(* IEC 61131-3 sources: example-modbus-rtu/PC WORX/export-st, 14 files *)

(* ---- sys_flag_types.IEC ---- *)
(*@PROPERTIES_EX@
TYPE: DATA_TYPE
LOCALE: 0
*)
TYPE
    Task_Name_Typ : ARRAY[0..9] OF BYTE;

    Extended_Task_Info : STRUCT
	    TaskName           : Task_Name_Typ;  (* Name of the Task as ARRAY OF BYTE, NULL terminated *)
	    TaskPrio           : INT;            (* Priority of the task *)
	    undocumented_0     : INT;
	    TaskPeriod         : INT;            (* Period of the task in milliseconds *)
	    TaskStack          : INT;            (* Stack size of the task *)
	    unused_1           : INT;
	    TaskWatchdog       : INT;            (* Watchdog time in milliseconds *)
	    undocumented_2     : INT;
	    undocumented_3     : INT;
	    undocumented_4     : INT;
	    CurDuration        : INT;            (* Current task duration in ticks including preemption *)
	    MinDuration        : INT;            (* Minimum task duration in ticks including preemption *)
	    MaxDuration        : INT;            (* Maximum task duration in ticks including preemption *)
	    undocumented_5     : INT;
	    CurDelay           : INT;            (* Current task delay in ticks including preemption *)
	    MinDelay           : INT;            (* Minimum task delay in ticks including preemption *)
	    MaxDelay           : INT;            (* Maximum task delay in ticks including preemption *)
    END_STRUCT;
END_TYPE

TYPE
	Task_Name_eCLR : ARRAY[0..35] OF BYTE;

	Task_Info_eCLR : STRUCT
		TaskStack       : INT;            (* Stack size of the task *)
		TaskPrio        : INT;            (* Priority of the task *)
		TaskPeriod_us   : DINT;           (* Period of the task in microseconds *)
		TaskWatchdog_us : DINT;           (* Watchdog time in microseconds *)
		TaskPeriod      : INT;            (* Period of the task in milliseconds *)
		TaskWatchdog    : INT;            (* Watchdog time in milliseconds *)
		MinDuration_us  : DINT;           (* Minimum task duration in microseconds including preemption *)
		MaxDuration_us  : DINT;           (* Maximum task duration in microseconds including preemption *)
		CurDuration_us  : DINT;           (* Current task duration in microseconds including preemption *)
		MinDelay_us     : DINT;           (* Minimum task delay in microseconds including preemption *)
		MaxDelay_us     : DINT;           (* Maximum task delay in microseconds including preemption *)
		CurDelay_us     : DINT;           (* Current task delay in microseconds including preemption *)
		MinDuration     : INT;            (* Minimum task duration in milliseconds including preemption *)
		MaxDuration     : INT;            (* Maximum task duration in milliseconds including preemption *)
		CurDuration     : INT;            (* Current task duration in milliseconds including preemption *)
		MinDelay        : INT;            (* Minimum task delay in milliseconds including preemption *)
		MaxDelay        : INT;            (* Maximum task delay in milliseconds including preemption *)
		CurDelay        : INT;            (* Current task delay in milliseconds including preemption *)
		unused_1        : DINT;
		unused_2        : DINT;
		unused_3        : DINT;
		unused_4        : DINT;
		unused_5        : DINT;
		unused_6        : DINT;
		unused_7        : DINT;
		unused_8        : DINT;
		unused_9        : DINT;
		TNameMaxSize    : INT;
		TNameSize       : INT;
		TaskName        : Task_Name_eCLR;
	END_STRUCT;
END_TYPE

TYPE
	PND_IO_6   : ARRAY[0..5]   OF BYTE;
	PND_IO_7   : ARRAY[0..6]   OF BYTE;
	PND_IO_32  : ARRAY[0..31]  OF BYTE;
	PND_IO_64  : ARRAY[0..63]  OF BYTE;
	PND_IO_128 : ARRAY[0..127] OF BYTE;
	PND_IO_256 : ARRAY[0..255] OF BYTE;
	PND_IO_512 : ARRAY[0..511] OF BYTE;
END_TYPE

TYPE
	Redundancy_OPC_Struct : ARRAY[0..2] OF INT;
END_TYPE

TYPE
    MBT_STATION_DIAG : STRUCT
	    Status           : DWORD; (* Bit 0 = Station is online*)
	                              (* Bit 1 = Exception exits  *)

	    IP               : DWORD;
	    OfflineCounter   : DWORD; (* Incremented by every shutdown of this station. *)

	    NetCycleAvg      : DWORD; (* ms. NetInCycleAvg + NetOutCycleAvg *)
	    NetCycleMin      : DWORD; (* ms. *)
	    NetCycleMax      : DWORD; (* ms. *)

	    NetInCycleAvg    : DWORD; (* ms. *)
	    NetInCycleMin    : DWORD; (* ms. *)
	    NetInCycleMax    : DWORD; (* ms. *)

	    NetOutCycleAvg   : DWORD; (* ms. *)
	    NetOutCycleMin   : DWORD; (* ms. *)
	    NetOutCycleMax   : DWORD; (* ms. *)

	    InternalError1   : DWORD; (* For internal use of Phoenix Contact! *)
	    InternalError2   : DWORD; (* For internal use of Phoenix Contact! *)

	    ExceptionCounter : DWORD; (* Incremented by every Modbus exception received on this station. *)
	    DiagReserved1    : BYTE;  (* Reserved for a later use! *)
	    DiagReserved2    : BYTE;  (* Reserved for a later use! *)
	    UnitID           : BYTE;  (* Modbus Unit Identifier *)
	    DiagReserved3    : BYTE;  (* Reserved for a later use! *)
    END_STRUCT;

    MBT_STATION_CONTROL : STRUCT
	    ctrlStatistics      : BYTE;  (* Bit 0 = Clear  statistics *)
	    ControlReserved1    : BYTE;  (* Reserved for a later use! *)
	    ControlReserved2    : WORD;  (* Reserved for a later use! *)
	    ControlReserved3    : DWORD; (* Reserved for a later use! *)
    END_STRUCT;
END_TYPE

TYPE
	MBS_SERVER_STATUS : STRUCT
		AcceptCnt              : DWORD;
		AcceptErrorCnt         : DWORD;
		ReceiveErrorCnt        : DWORD;
		ModbusRequestCnt       : DWORD;
		ModbusExceptionCnt     : DWORD;

		SocketErrorCode        : WORD;
		TcpConnectedClients    : WORD;
		LastExceptionRegister  : WORD;
		LastExceptionRegLength : WORD;

		LastExceptionNode      : BYTE;
		LastExceptionFunction  : BYTE;
		LastExceptionCode      : BYTE;
		reserved               : BYTE;
	END_STRUCT;
END_TYPE

TYPE
	MBS_SERVER_CONTROL : STRUCT
		Flags     : BYTE;
		reserved1 : BYTE;
		reserved2 : BYTE;
		reserved3 : BYTE;
	END_STRUCT;
END_TYPE

TYPE
	MBS_NODE_STATUS : STRUCT
		ModbusRequestCnt   : DWORD;
		ModbusExceptionCnt : DWORD;
		Flags              : DWORD;
		reserved           : DWORD;
	END_STRUCT;
END_TYPE

TYPE
    OPCUA_STATUS_INFO : STRUCT
	  restartCount            : UDINT; (* each reset and clear cache is counted *)
	  monitoredVariablesCount : UDINT; (* use IdataSource.GetSubscribedVariablesCount *)
	  sessionsCount           : UDINT; (* <-- get Data from ServerDiagnostic method GetTotalSubscribedVariablesCount *)
	  isServerEnabled         : UDINT; (* fetched by conf API *)
	  isLicensePresent        : UDINT; (* fetched by lic API *)
	END_STRUCT;
END_TYPE

TYPE
    IEC61850_TIMESTAMP : STRUCT
	    Seconds     : DWORD;
		Fractions   : DWORD;
        TimeQuality : DWORD;
    END_STRUCT;
END_TYPE

TYPE
	PROFISAFE_DIAG_HEADER : STRUCT
		NumberOfFConn         : UINT; (* number of F-Connections, max 256 *)
		PLCHostStatusByte     : BYTE; (* status byte of Standard PLC *)
		SPNSAgentStatusByte   : BYTE; (* status byte of SPNS agent *)
		CycleCount            : UINT;   (* cycle count off the spns agent (update the shm diag area) *)
	END_STRUCT;

	F_MESSAGE : ARRAY[0..15] OF BYTE; (* F-message: 16 bytes *)

	F_DEVICE_DIAG : STRUCT
		FAddress     : WORD;      (* F address of device  *)
		F_WD_Time    : WORD;      (* F WD time of device  *)
		F_DataLenIn  : BYTE;      (* length of IN F data  *)
		F_MessageIn  : F_MESSAGE; (* IN F data array      *)
		F_DataLenOut : BYTE;      (* length of OUT F data *)
		F_MessageOut : F_MESSAGE; (* OUT F data array     *)
	END_STRUCT;

	DEVICE_DIAG_LIST : ARRAY[0..255] OF F_DEVICE_DIAG; (* array of F_DEVICE_DIAG structurs: 256 elem *)

	PROFISAFE_DIAG : STRUCT
		ProfisafeDiagHeader : PROFISAFE_DIAG_HEADER; (* header *)
		FDeviceDiagnostics  : DEVICE_DIAG_LIST;      (* list of diagnostics *)
	END_STRUCT;
END_TYPE

TYPE
	PROFISAFE_RECORD : STRUCT
	   	CodeName              : DWORD;                   (* F_S/D_Address *)
   		ProfiSafeDiagBitField : DWORD;
   		SrtMin                : UINT;                    (* minimal safety round trip time of the connection *)
   		SrtMax                : UINT;                    (* maximal safety round trip time of the connection *)
   		SrtCur                : UINT;                    (* current safety round trip time of the connection *)
   		FWdTime               : UINT;                    (* parameterized f-wd-time *)
   		ValidReg              : UINT;                    (* the values in this profisafe record are balid or not *)
      	Reserved              : UINT;                    (* to fill up the structure to a size x*4 *)
 	END_STRUCT;

    PROFISAFE_RECORD_ARRAY : ARRAY[0..299] OF PROFISAFE_RECORD;

    PROFISAFE_DIAG_OUT : STRUCT
   		MaxNumberOfProfiSafeRecords : UINT; (* max. number of possible profisafe records *)
   		NumberOfProfiSafeRecords    : UINT; (* current number of possible profisafe records in array *)
   		ProfiSafeRecord             : PROFISAFE_RECORD_ARRAY;
   		ProfiSafeGlobalRecord       : DWORD;
 	END_STRUCT;
END_TYPE

(* ---- udtModbusControl.IEC ---- *)
(*@PROPERTIES_EX@
TYPE: DATA_TYPE
LOCALE: 0
*)
TYPE
	udtModbusControl	:
	STRUCT
		(* Commands to Modbus FB *)
		uiSlaveAddress		: UINT;

		xSendRequest_FC3	: BOOL;
		uiStartAddress_FC3	: UINT;
		iDataCount_FC3		: INT;

		xSendRequest_FC4	: BOOL;
		uiStartAddress_FC4	: UINT;
		iDataCount_FC4		: INT;

		xSendRequest_FC6	: BOOL;
		uiStartAddress_FC6	: UINT;

		(* Data from Modbus FB *)
		xDone_FC3			: BOOL;
		xError_FC3			: BOOL;
		arrReadData_FC3		: arrModbus2_W_1_125;

		xDone_FC4			: BOOL;
		xError_FC4			: BOOL;
		arrReadData_FC4		: arrModbus2_W_1_125;

		xDone_FC6			: BOOL;
		xError_FC6			: BOOL;
		wValue_FC6			: WORD;

		(* From udtMaster structure *)
		Master_uiRcvDataCount	: UINT;
		Master_uiSlaveAddress	: UINT;
		Master_uiStartAddress	: UINT;
		Master_iFunctionCode	: INT;
	END_STRUCT;
END_TYPE

(* ---- udtModbusDevice.IEC ---- *)
(*@PROPERTIES_EX@
TYPE: DATA_TYPE
LOCALE: 0
*)
TYPE
	udtModbusDiagValues:
	STRUCT
		xError							: BOOL;
		wDiagCode						: WORD;
		strDiagCode						: STRING;
	END_STRUCT;

	udtModbusConfiguration:
	STRUCT
		uiSlaveAddress					: UINT;
	END_STRUCT;

	udtDeviceConfiguration:
	STRUCT
		Modbus							: udtModbusConfiguration;
	END_STRUCT;

	udtDeviceDiagValues:
	STRUCT
		xError							: BOOL;
		wDiagCode						: WORD;
		strDiagCode						: STRING;

		Modbus							: udtModbusDiagValues;
	END_STRUCT;

	udtModbusDeviceValues:
	STRUCT
		iRtcMinutes						: INT;
	END_STRUCT;

	udtModbusDevice:
	STRUCT
		Configuration					: udtDeviceConfiguration;
		DataValues						: udtModbusDeviceValues;
		DiagValues						: udtDeviceDiagValues;
	END_STRUCT;
END_TYPE

(* ---- ErrorHandler.ST ---- *)
(*@PROPERTIES_EX@
TYPE: POU
LOCALE: 0
IEC_LANGUAGE: ST
PLC_TYPE: independent
PROC_TYPE: independent
GROUP: Modbus
*)
(*@KEY@:DESCRIPTION*)

(*@KEY@:END_DESCRIPTION*)
FUNCTION_BLOCK ErrorHandler

(*Group:Default*)

VAR_INPUT
	xError :	BOOL;
END_VAR

VAR
	wLastDiagCode :	WORD;
	wLastAddDiagCode :	WORD;
END_VAR

VAR_INPUT
	wDiagCode :	WORD;
	wAddDiagCode :	WORD;
END_VAR

(*@KEY@: WORKSHEET
NAME: ErrorHandler
IEC_LANGUAGE: ST
*)
IF xError THEN

	wLastDiagCode := wDiagCode;
	wLastAddDiagCode := wAddDiagCode;

END_IF;
(*@KEY@: END_WORKSHEET *)
END_FUNCTION_BLOCK

(* ---- MB_RTU_FC3_ABSTRACT.ST ---- *)
(*@PROPERTIES_EX@
TYPE: POU
LOCALE: 0
IEC_LANGUAGE: ST
PLC_TYPE: independent
PROC_TYPE: independent
GROUP: Modbus
*)
(*@KEY@:DESCRIPTION*)

(*@KEY@:END_DESCRIPTION*)
FUNCTION_BLOCK MB_RTU_FC3_ABSTRACT

(*Group:Input*)

VAR_INPUT
	xActivate :	BOOL;
	xSendRequest :	BOOL;
	xTimeout :	BOOL;
	uiSlaveAddress :	UINT;
	uiStartAddress :	UINT;
	iDataCount :	INT;
END_VAR

(*Group:Output*)

VAR_OUTPUT
	xDone :	BOOL;
	xError :	BOOL;
	xBusy :	BOOL;
	arrReadData :	arrModbus2_W_1_125;
END_VAR

(*Group:Inout*)

VAR_IN_OUT
	udtModbusControl :	udtModbusControl;
END_VAR

(*Group:Default*)

VAR
	iStep :	INT;
END_VAR

(*@KEY@: WORKSHEET
NAME: MB_RTU_FC3_ABSTRACT
IEC_LANGUAGE: ST
*)
IF xActivate THEN

	CASE iStep OF

		0:

			xDone	:= FALSE;
			xError	:= FALSE;

			IF xSendRequest THEN

				udtModbusControl.iDataCount_FC3 		:= iDataCount;
				udtModbusControl.uiSlaveAddress 		:= uiSlaveAddress;
				udtModbusControl.uiStartAddress_FC3		:= uiStartAddress;
				udtModbusControl.xSendRequest_FC3		:= TRUE;

				xBusy	:= TRUE;

				iStep := 1;

			END_IF;

		1:

	      udtModbusControl.xSendRequest_FC3     := FALSE;
		  udtModbusControl.iDataCount_FC3 		:= iDataCount;
		  udtModbusControl.uiSlaveAddress 		:= uiSlaveAddress;
		  udtModbusControl.uiStartAddress_FC3	:= uiStartAddress;

	      IF 	((udtModbusControl.xDone_FC3 OR
	        	udtModbusControl.xError_FC3) AND
	      		(udtModbusControl.Master_uiRcvDataCount = INT_TO_UINT(iDataCount * 2)) AND
	      		(udtModbusControl.Master_uiSlaveAddress  = uiSlaveAddress) AND
	      		(udtModbusControl.Master_uiStartAddress = uiStartAddress) AND
	      		(udtModbusControl.Master_iFunctionCode = 3))

				OR

				(*
				(xTimeout AND
				(udtModbusControl.Master_uiSlaveAddress  = uiSlaveAddress) AND
	      		(udtModbusControl.Master_uiStartAddress = uiStartAddress) AND
	      		(udtModbusControl.Master_iFunctionCode = 3))
				*)

				xTimeout

		  	THEN

					IF udtModbusControl.xDone_FC3 THEN
						arrReadData := udtModbusControl.arrReadData_FC3;
					END_IF;

					xDone	:= udtModbusControl.xDone_FC3;
					xError	:= udtModbusControl.xError_FC3 OR xTimeout;

					xBusy	:= FALSE;

					iStep := 0;

				END_IF;

	END_CASE;

ELSE

	xDone	:= FALSE;
	xError	:= FALSE;
	xBusy	:= FALSE;
	iStep	:= 0;

END_IF;

(*@KEY@: END_WORKSHEET *)
END_FUNCTION_BLOCK

(* ---- MB_RTU_FC4_ABSTRACT.ST ---- *)
(*@PROPERTIES_EX@
TYPE: POU
LOCALE: 0
IEC_LANGUAGE: ST
PLC_TYPE: independent
PROC_TYPE: independent
GROUP: Modbus
*)
(*@KEY@:DESCRIPTION*)

(*@KEY@:END_DESCRIPTION*)
FUNCTION_BLOCK MB_RTU_FC4_ABSTRACT

(*Group:Input*)

VAR_INPUT
	xActivate :	BOOL;
	xSendRequest :	BOOL;
	xTimeout :	BOOL;
	uiSlaveAddress :	UINT;
	uiStartAddress :	UINT;
	iDataCount :	INT;
END_VAR

(*Group:Output*)

VAR_OUTPUT
	xDone :	BOOL;
	xError :	BOOL;
	xBusy :	BOOL;
	arrReadData :	arrModbus2_W_1_125;
END_VAR

(*Group:Inout*)

VAR_IN_OUT
	udtModbusControl :	udtModbusControl;
END_VAR

(*Group:Default*)

VAR
	iStep :	INT;
END_VAR

(*@KEY@: WORKSHEET
NAME: MB_RTU_FC4_ABSTRACT
IEC_LANGUAGE: ST
*)
IF xActivate THEN

	CASE iStep OF

		0:

			xDone	:= FALSE;
			xError	:= FALSE;

			IF xSendRequest THEN

				udtModbusControl.iDataCount_FC4 		:= iDataCount;
				udtModbusControl.uiSlaveAddress 		:= uiSlaveAddress;
				udtModbusControl.uiStartAddress_FC4		:= uiStartAddress;
				udtModbusControl.xSendRequest_FC4		:= TRUE;

				xBusy	:= TRUE;

				iStep := 1;

			END_IF;

		1:

	      udtModbusControl.xSendRequest_FC4     := FALSE;
		  udtModbusControl.iDataCount_FC4 		:= iDataCount;
		  udtModbusControl.uiSlaveAddress 		:= uiSlaveAddress;
		  udtModbusControl.uiStartAddress_FC4	:= uiStartAddress;

	      IF 	((udtModbusControl.xDone_FC4 OR
	        	udtModbusControl.xError_FC4) AND
	      		(udtModbusControl.Master_uiRcvDataCount = INT_TO_UINT(iDataCount * 2)) AND
	      		(udtModbusControl.Master_uiSlaveAddress  = uiSlaveAddress) AND
	      		(udtModbusControl.Master_uiStartAddress = uiStartAddress) AND
	      		(udtModbusControl.Master_iFunctionCode = 4))

				OR

				(*
				(xTimeout AND
				(udtModbusControl.Master_uiSlaveAddress  = uiSlaveAddress) AND
	      		(udtModbusControl.Master_uiStartAddress = uiStartAddress) AND
	      		(udtModbusControl.Master_iFunctionCode = 3))
				*)

				xTimeout

		  	THEN

					IF udtModbusControl.xDone_FC4 THEN
						arrReadData := udtModbusControl.arrReadData_FC4;
					END_IF;

					xDone	:= udtModbusControl.xDone_FC4;
					xError	:= udtModbusControl.xError_FC4 OR xTimeout;

					xBusy	:= FALSE;

					iStep := 0;

				END_IF;

	END_CASE;

ELSE

	xDone	:= FALSE;
	xError	:= FALSE;
	xBusy	:= FALSE;
	iStep	:= 0;

END_IF;

(*@KEY@: END_WORKSHEET *)
END_FUNCTION_BLOCK

(* ---- MB_RTU_FC6_ABSTRACT.ST ---- *)
(*@PROPERTIES_EX@
TYPE: POU
LOCALE: 0
IEC_LANGUAGE: ST
PLC_TYPE: independent
PROC_TYPE: independent
GROUP: Modbus
*)
(*@KEY@:DESCRIPTION*)

(*@KEY@:END_DESCRIPTION*)
FUNCTION_BLOCK MB_RTU_FC6_ABSTRACT

(*Group:Default*)

VAR
	iStep :	INT;
END_VAR

(*Group:Input*)

VAR_INPUT
	xActivate :	BOOL;
	xSendRequest :	BOOL;
	xTimeout :	BOOL;
	uiSlaveAddress :	UINT;
	uiStartAddress :	UINT;
	wValue :	WORD;
END_VAR

(*Group:Output*)

VAR_OUTPUT
	xDone :	BOOL;
	xError :	BOOL;
	xBusy :	BOOL;
END_VAR

(*Group:Inout*)

VAR_IN_OUT
	udtModbusControl :	udtModbusControl;
END_VAR

(*@KEY@: WORKSHEET
NAME: MB_RTU_FC6_ABSTRACT
IEC_LANGUAGE: ST
*)
IF xActivate THEN

	CASE iStep OF

		0:

			xDone	:= FALSE;
			xError	:= FALSE;

			IF xSendRequest THEN

				udtModbusControl.uiSlaveAddress 		:= uiSlaveAddress;
				udtModbusControl.uiStartAddress_FC6		:= uiStartAddress;
				udtModbusControl.wValue_FC6				:= wValue;
				udtModbusControl.xSendRequest_FC6		:= TRUE;

				xBusy	:= TRUE;

				iStep := 1;

			END_IF;

		1:

			udtModbusControl.xSendRequest_FC6      := FALSE;
			udtModbusControl.uiSlaveAddress 		:= uiSlaveAddress;
			udtModbusControl.uiStartAddress_FC6		:= uiStartAddress;
			udtModbusControl.wValue_FC6				:= wValue;

			IF 	(
				(udtModbusControl.xDone_FC6 OR
	        	udtModbusControl.xError_FC6) AND
	      		(udtModbusControl.Master_uiSlaveAddress  = uiSlaveAddress) AND
	      		(udtModbusControl.Master_uiStartAddress = uiStartAddress) AND
	      		(udtModbusControl.Master_iFunctionCode = 6)
				)
				OR
				xTimeout

		  	THEN

					xDone	:= udtModbusControl.xDone_FC6;
					xError	:= udtModbusControl.xError_FC6 OR xTimeout;

					xBusy	:= FALSE;

					iStep := 0;

				END_IF;

	END_CASE;

ELSE

	xDone	:= FALSE;
	xError	:= FALSE;
	xBusy	:= FALSE;
	iStep	:= 0;

END_IF;

(*@KEY@: END_WORKSHEET *)
END_FUNCTION_BLOCK

(* ---- ModbusDeviceHandler.ST ---- *)
(*@PROPERTIES_EX@
TYPE: POU
LOCALE: 0
IEC_LANGUAGE: ST
PLC_TYPE: independent
PROC_TYPE: independent
GROUP: Modbus
*)
(*@KEY@:DESCRIPTION*)

(*@KEY@:END_DESCRIPTION*)
FUNCTION_BLOCK ModbusDeviceHandler

(*Group:POU`s*)

VAR
	TIME_DIFF :	TIME_DIFF;
	REQUEST_ERROR :	REQUEST_ERROR;
	MB_RTU_FC3_ABSTRACT :	MB_RTU_FC3_ABSTRACT;
END_VAR

(*Group:INTERNAL*)

VAR
	arrReadData_FC3 :	arrModbus2_W_1_125;
	xBusy_FC3 :	BOOL;
	xDone_FC3 :	BOOL;
	xError_FC3 :	BOOL;
	xTimeout_FC3 :	BOOL;
END_VAR

(*Group:INPUT*)

VAR_INPUT
	xActivate :	BOOL;
	xSendRequest_IN :	BOOL;
	uiSlaveAddress :	UINT;
END_VAR

(*Group:OUTPUT*)

VAR_OUTPUT
	xConnectionBroken :	BOOL;
	diTimeDiff :	DINT;
	xSendRequest_OUT :	BOOL;
END_VAR

(*Group:IN - OUT*)

VAR_INPUT
	ModbusDeviceData :	udtModbusDevice;
END_VAR

VAR_IN_OUT
	udtModbusControl :	udtModbusControl;
END_VAR

(*Group:Default*)

VAR_INPUT
	tTimeout :	TIME;
END_VAR

VAR
	RS_REQUEST_IN_PROGRESS :	RS;
END_VAR

(*@KEY@: WORKSHEET
NAME: ModbusDeviceHandler
IEC_LANGUAGE: ST
*)
(*	Request in progress *)
RS_REQUEST_IN_PROGRESS.SET					:= xActivate AND xSendRequest_IN;
RS_REQUEST_IN_PROGRESS.RESET1				:= NOT xActivate OR (xDone_FC3 OR xError_FC3);
RS_REQUEST_IN_PROGRESS();

(*	FC 3 *)
MB_RTU_FC3_ABSTRACT.xActivate				:= xActivate;
MB_RTU_FC3_ABSTRACT.xSendRequest			:= RS_REQUEST_IN_PROGRESS.Q1;
MB_RTU_FC3_ABSTRACT.xTimeout				:= xTimeout_FC3;
MB_RTU_FC3_ABSTRACT.uiSlaveAddress			:= uiSlaveAddress;
MB_RTU_FC3_ABSTRACT.uiStartAddress			:= UINT#1;
MB_RTU_FC3_ABSTRACT.iDataCount				:= INT#1;
MB_RTU_FC3_ABSTRACT.udtModbusControl		:= udtModbusControl;

MB_RTU_FC3_ABSTRACT();

xDone_FC3									:= MB_RTU_FC3_ABSTRACT.xDone;
xError_FC3									:= MB_RTU_FC3_ABSTRACT.xError;
xBusy_FC3									:= MB_RTU_FC3_ABSTRACT.xBusy;
arrReadData_FC3								:= MB_RTU_FC3_ABSTRACT.arrReadData;
udtModbusControl							:= MB_RTU_FC3_ABSTRACT.udtModbusControl;

(*	Pass the request to the next device handler *)
xSendRequest_OUT							:= RS_REQUEST_IN_PROGRESS.Q1 AND (xDone_FC3 OR xError_FC3);

(*	Detect errors *)
REQUEST_ERROR.xReq							:= xBusy_FC3;
REQUEST_ERROR.xDone							:= xDone_FC3;
REQUEST_ERROR.xError						:= xError_FC3;
REQUEST_ERROR.iMaxErrorCnt					:= 5;
REQUEST_ERROR.tTimeout						:= tTimeout;

REQUEST_ERROR();

xTimeout_FC3								:= REQUEST_ERROR.xTimeout;
ModbusDeviceData.DiagValues.Modbus.xError	:= REQUEST_ERROR.xConnectBroken;
xConnectionBroken							:= REQUEST_ERROR.xConnectBroken;

(*	Measure request time *)
TIME_DIFF.xIN1								:= xSendRequest_IN;
TIME_DIFF.xIN2								:= xSendRequest_OUT;
TIME_DIFF();
diTimeDiff									:= TIME_DIFF.diSystemTickDiff;

(*	Handle data values *)
ModbusDeviceData.DataValues.iRtcMinutes		:= WORD_TO_INT(arrReadData_FC3[1]);

(*	Handle diag values *)
IF ModbusDeviceData.DiagValues.Modbus.xError THEN

	ModbusDeviceData.DiagValues.xError		:=	TRUE;
	ModbusDeviceData.DiagValues.strDiagCode	:=	'RS-485 connection error';

ELSE
	ModbusDeviceData.DiagValues.xError		:=	FALSE;
	ModbusDeviceData.DiagValues.strDiagCode	:=	'OK';
END_IF;

(*@KEY@: END_WORKSHEET *)
END_FUNCTION_BLOCK

(* ---- REQ_CNT.ST ---- *)
(*@PROPERTIES_EX@
TYPE: POU
LOCALE: 0
IEC_LANGUAGE: ST
PLC_TYPE: independent
PROC_TYPE: independent
GROUP: Modbus
*)
(*@KEY@:DESCRIPTION*)
(*
FB generate a boolean output if:
	uiReqNo
	uiRespNo
do not counting up longer than specified delay time

*)
************
Versioning
************

15.01.2016	KONOPKOV Inital Version

(*@KEY@:END_DESCRIPTION*)
FUNCTION_BLOCK REQ_CNT

(*Group:outputs*)

VAR_OUTPUT
	xOut :	BOOL;
END_VAR

(*Group:internal*)

VAR
	uiReqNo_Registered :	UINT {RDT};
	uiRespNo_Registered :	UINT {RDT};
	TON_1 :	TON;
	TON_2 :	TON;
END_VAR

(*Group:inputs*)

VAR_INPUT
	xDisable :	BOOL;
	tTimeDelayRequests :	TIME;
	tTimeDelayResponces :	TIME;
	uiReqNo :	UINT;
	uiRespNo :	UINT;
END_VAR

VAR
	R_TRIG_1 :	R_TRIG;
END_VAR

(*@KEY@: WORKSHEET
NAME: REQ_CNT
IEC_LANGUAGE: ST
*)
(*
FB generate a boolean output if:
	uiReqNo
	uiRespNo
do not counting up longer than specified delay time

*)

TON_1.IN := (uiReqNo = uiReqNo_Registered AND NOT xDisable AND NOT xOut);
TON_1.PT := tTimeDelayRequests;
TON_1(); (*uiReqNo*)

TON_2.IN := (uiRespNo = uiRespNo_Registered AND NOT xDisable AND NOT xOut);
TON_2.PT := tTimeDelayResponces;
TON_2(); (*uiRespNo*)

R_TRIG_1.CLK 	:= TON_1.Q OR TON_2.Q;
R_TRIG_1();
xOut			:= R_TRIG_1.Q;

IF uiReqNo <> uiReqNo_Registered THEN
	uiReqNo_Registered := uiReqNo;
END_IF;

IF uiRespNo <> uiRespNo_Registered THEN
	uiRespNo_Registered := uiRespNo;
END_IF;

(*@KEY@: END_WORKSHEET *)
END_FUNCTION_BLOCK

(* ---- REQUEST_ERROR.ST ---- *)
(*@PROPERTIES_EX@
TYPE: POU
LOCALE: 0
IEC_LANGUAGE: ST
PLC_TYPE: independent
PROC_TYPE: independent
GROUP: Modbus
*)
(*@KEY@:DESCRIPTION*)
**************************************************************************

Copyright © 2016 Phoenix Contact Russia
All rights reserved

**************************************************************************
Name	:	 REQUEST_ERROR

State	:	[ ] evaluation  [x] released

Develop Environment	:
	PC WORX 	:	6.30.1668 (AX SW Suite 2016 Hotfix1)
	Controller	:	AXC 1050 FW v2.10
	Devices		: 	No

**************************************************************************

Change Notes:

Date		Version		Author		Description
--------------------------------------------------------------------------
08.08.16	1.00		konopkov	initial version

**************************************************************************
Description:
Индикация ошибки отсутствия обмена данными при достижении заданного количества
импульсов на вход Ошибка.

(*@KEY@:END_DESCRIPTION*)
FUNCTION_BLOCK REQUEST_ERROR

(*Group:Input*)

VAR_INPUT
	xReq :	BOOL;(*???? ??????*)
	xDone :	BOOL;(*???? ????? ??*)
	xError :	BOOL;(*???? ????? ??????*)
	iMaxErrorCnt :	INT := 5;(*???????????? ?????????? ????????? ?????? ? ??????????? ??????????????????*)
	tTimeout :	TIME;
END_VAR

(*Group:Output*)

VAR_OUTPUT
	xConnectBroken :	BOOL;(*??????? ??????????????? ?????? ?????*)
	xTimeout :	BOOL;
END_VAR

(*Group:Internal*)

VAR_OUTPUT
	iErrorCnt :	INT;(*??????? ??????*)
END_VAR

(*Group:Instances*)

VAR
	R_TRIG_DONE :	R_TRIG;
	R_TRIG_ERROR :	R_TRIG;
	R_TRIG_REQUEST :	R_TRIG;
	RS_REQUEST :	RS;
	TON_REQUEST :	TON;
END_VAR

(*@KEY@: WORKSHEET
NAME: REQUEST_ERROR
IEC_LANGUAGE: ST
*)
(*
xConnectBroken
xDone
xError
iMaxErrorCnt
*)

IF R_TRIG_ERROR.Q OR TON_REQUEST.Q THEN
	iErrorCnt := iErrorCnt + 1;
END_IF;

IF R_TRIG_DONE.Q THEN
	iErrorCnt := 0;
END_IF;

IF iErrorCnt >= iMaxErrorCnt THEN
	xConnectBroken := TRUE;
ELSE
	xConnectBroken := FALSE;
END_IF;

R_TRIG_DONE(CLK:=xDone);
R_TRIG_ERROR(CLK:=xError);
R_TRIG_REQUEST(CLK:=xReq);

RS_REQUEST.SET 		:= R_TRIG_REQUEST.Q;
RS_REQUEST.RESET1	:= R_TRIG_DONE.Q OR R_TRIG_ERROR.Q OR TON_REQUEST.Q;
RS_REQUEST();

TON_REQUEST.IN		:= RS_REQUEST.Q1;
TON_REQUEST.PT		:= tTimeout;
TON_REQUEST();
xTimeout 			:= TON_REQUEST.Q;

(*@KEY@: END_WORKSHEET *)
END_FUNCTION_BLOCK

(* ---- SlaveDevice.ST ---- *)
(*@PROPERTIES_EX@
TYPE: POU
LOCALE: 0
IEC_LANGUAGE: ST
PLC_TYPE: independent
PROC_TYPE: independent
GROUP: Mock
*)
(*@KEY@:DESCRIPTION*)

(*@KEY@:END_DESCRIPTION*)
FUNCTION_BLOCK SlaveDevice

(*Group:Inouts*)

VAR_IN_OUT
	udtRS485Line :	udtRS485Frame;
END_VAR

(*Group:Inputs*)

VAR_INPUT
	xActivate :	BOOL;
	xDebug :	BOOL;
	strConsoleId :	STRING;
	uiSlaveAddress :	UINT := UINT#1;
END_VAR

(*Group:Mock*)

VAR
	IL_UNI07_Slave :	IL_UNI07;
END_VAR

(*Group:Global*)

VAR_EXTERNAL
	RTC_SECONDS :	INT;(*System time (seconds)*)
END_VAR

(*Group:Slave*)

VAR
	MB_IL_UNI07_Slave :	MB_IL_UNI07_Slave_3;
	udtHoldingRegisters :	arrModbus2_w_0_1999;
	udtInputRegisters :	arrModbus2_w_2000_2999;
	udtOutputBits :	arrModbus2_x_3000_3999;
	udtInputBits :	arrModbus2_x_4000_4999;
	arrInputAddressSlave :	MB2_RSUNI_ARR_B_1_14;
	arrOutputAddressSlave :	MB2_RSUNI_ARR_B_1_14;
END_VAR

(*@KEY@: WORKSHEET
NAME: SlaveDevice
IEC_LANGUAGE: ST
*)
(*	IB IL RS UNI (Proceess data 7 words) software replacement *)
IL_UNI07_Slave.xConsoleLog				:= xDebug;
IL_UNI07_Slave.strConsoleId				:= strConsoleId;
IL_UNI07_Slave.udtRS485Line				:= udtRS485Line;
IL_UNI07_Slave.arrInputAddress			:= arrOutputAddressSlave;
IL_UNI07_Slave.arrOutputAddress			:= arrInputAddressSlave;

IL_UNI07_Slave();

udtRS485Line							:= IL_UNI07_Slave.udtRS485Line;
arrOutputAddressSlave					:= IL_UNI07_Slave.arrInputAddress;
arrInputAddressSlave					:= IL_UNI07_Slave.arrOutputAddress;

(*
MB_Master block receives data from
mocked IB IL RS UNI function block instead of Process data
*)

MB_IL_UNI07_Slave.xActivate				:= xActivate;
MB_IL_UNI07_Slave.bSelectMode			:= BYTE#01;
MB_IL_UNI07_Slave.diBaudrate			:= DINT#9600;
MB_IL_UNI07_Slave.wDataWidth			:= WORD#4;
MB_IL_UNI07_Slave.uiSlaveAddress		:= uiSlaveAddress;
MB_IL_UNI07_Slave.udtHoldingRegisters	:= udtHoldingRegisters;
MB_IL_UNI07_Slave.udtInputRegisters		:= udtInputRegisters;
MB_IL_UNI07_Slave.udtOutputBits			:= udtOutputBits;
MB_IL_UNI07_Slave.udtInputBits			:= udtInputBits;
MB_IL_UNI07_Slave.arrInputAddress		:= arrInputAddressSlave;
MB_IL_UNI07_Slave.arrOutputAddress		:= arrOutputAddressSlave;

MB_IL_UNI07_Slave();

udtHoldingRegisters         			:= MB_IL_UNI07_Slave.udtHoldingRegisters;
udtInputRegisters           			:= MB_IL_UNI07_Slave.udtInputRegisters;
udtOutputBits           				:= MB_IL_UNI07_Slave.udtOutputBits;
udtInputBits            				:= MB_IL_UNI07_Slave.udtInputBits;
arrInputAddressSlave            		:= MB_IL_UNI07_Slave.arrInputAddress;
arrOutputAddressSlave           		:= MB_IL_UNI07_Slave.arrOutputAddress;

(*	Fill in register value *)
udtHoldingRegisters[1]					:= INT_TO_WORD(100 * UINT_TO_INT(uiSlaveAddress)+ RTC_SECONDS);

(*@KEY@: END_WORKSHEET *)
END_FUNCTION_BLOCK

(* ---- TIME_DIFF.ST ---- *)
(*@PROPERTIES_EX@
TYPE: POU
LOCALE: 0
IEC_LANGUAGE: ST
PLC_TYPE: independent
PROC_TYPE: independent
GROUP: Modbus
*)
(*@KEY@:DESCRIPTION*)

(*@KEY@:END_DESCRIPTION*)
FUNCTION_BLOCK TIME_DIFF

(*Group:Default*)

VAR_INPUT
	xReset :	BOOL;
	xIN1 :	BOOL;
	xIN2 :	BOOL;
END_VAR

VAR_OUTPUT
	diSystemTickDiff :	DINT;
END_VAR

VAR
	diSystemTick_IN1 :	DINT;
	diSystemTick_IN2 :	DINT;
	R_TRIG_1 :	R_TRIG;
	R_TRIG_2 :	R_TRIG;
	R_TRIG_3 :	R_TRIG;
END_VAR

VAR_EXTERNAL
	PLC_SYS_TICK_CNT :	DINT;(*Number of system ticks*)
END_VAR

(*@KEY@: WORKSHEET
NAME: TIME_DIFF
IEC_LANGUAGE: ST
*)
R_TRIG_1(CLK:=xIN1);

R_TRIG_2(CLK:=xIN2);

R_TRIG_3(CLK:=xReset);

IF R_TRIG_1.Q THEN
	diSystemTick_IN1 := PLC_SYS_TICK_CNT;
END_IF;

IF R_TRIG_2.Q THEN
	diSystemTick_IN2 := PLC_SYS_TICK_CNT;
	diSystemTickDiff := diSystemTick_IN2 - diSystemTick_IN1;
END_IF;

IF R_TRIG_3.Q THEN
	diSystemTick_IN1 := DINT#0;
	diSystemTick_IN2 := DINT#0;
	diSystemTickDiff := DINT#0;
END_IF;

(*@KEY@: END_WORKSHEET *)
END_FUNCTION_BLOCK

(* ---- Main.ST ---- *)
(*@PROPERTIES_EX@
TYPE: POU
LOCALE: 0
IEC_LANGUAGE: ST
PLC_TYPE: independent
PROC_TYPE: independent
*)
(*@KEY@:DESCRIPTION*)

(*@KEY@:END_DESCRIPTION*)
PROGRAM Main

(*Group:Master*)

VAR
	MB_IL_UNI07_Master :	MB_IL_UNI07_Master_5;
	MB_RTU_FC3 :	MB_RTU_FC3_5;
	R_TRIG_MASTER_ACTIVE :	R_TRIG;
	xActivateMaster :	BOOL := TRUE;
	xResetMaster :	BOOL;
	udtMbDataMaster :	udtModbus2_Data;
	arrInputAddressMaster :	MB2_RSUNI_ARR_B_1_14;
	arrOutputAddressMaster :	MB2_RSUNI_ARR_B_1_14;
	wDiagCodeFC3 :	WORD;
	wAddDiagCodeFC3 :	WORD;
	xStartOfPoll :	BOOL;
	xEndOfPoll :	BOOL;
END_VAR

(*Group:Global*)

VAR_EXTERNAL
	udtRS485Line :	udtRS485Frame;
END_VAR

VAR
	MB_RTU_FC6 :	MB_RTU_FC6_5;
	REQ_CNT :	REQ_CNT;
	ModbusControl :	udtModbusControl;
END_VAR

(*Group:Slave handlers*)

VAR
	xActivate01 :	BOOL := TRUE;
	ModbusDeviceHandler01 :	ModbusDeviceHandler;
	ModbusDeviceData01 :	udtModbusDevice;
	xConnectionBroken01 :	BOOL;
	diTimeDiff01 :	DINT;
	iRtcData01 :	INT;
	xActivate02 :	BOOL := TRUE;
	ModbusDeviceHandler02 :	ModbusDeviceHandler;
	ModbusDeviceData02 :	udtModbusDevice;
	xConnectionBroken02 :	BOOL;
	diTimeDiff02 :	DINT;
	iRtcData02 :	INT;
END_VAR

(*Group:Mock*)

VAR
	xDebug :	BOOL;
	IB_IL_RS_UNI_07_Master :	IL_UNI07;
END_VAR

(*@KEY@: WORKSHEET
NAME: Master
IEC_LANGUAGE: ST
*)
(*	Detect if Responce or Request Counters are not incrementing, and re-activate Master block *)
REQ_CNT.tTimeDelayRequests				:= T#5S;
REQ_CNT.tTimeDelayResponces				:= T#30S;
REQ_CNT.uiReqNo							:= MB_IL_UNI07_Master.uiRequestsCounter;
REQ_CNT.uiRespNo						:= MB_IL_UNI07_Master.uiResponsesCounter;

REQ_CNT();

xActivateMaster							:= NOT REQ_CNT.xOut;

(*	Start of request to first device in a line *)
xStartOfPoll							:= R_TRIG_MASTER_ACTIVE.Q OR xEndOfPoll;

R_TRIG_MASTER_ACTIVE.CLK				:= MB_IL_UNI07_Master.xActive;
R_TRIG_MASTER_ACTIVE();

(*
MB_Master block sends data to
mocked IB IL RS UNI function block instead of Process data
*)

MB_IL_UNI07_Master.xActivate			:= xActivateMaster;
MB_IL_UNI07_Master.bSelectMode			:= BYTE#01;
MB_IL_UNI07_Master.diBaudrate			:= DINT#9600;
MB_IL_UNI07_Master.wDataWidth			:= WORD#4;
MB_IL_UNI07_Master.tTimeout				:= T#1S;
MB_IL_UNI07_Master.xReset				:= xResetMaster;
MB_IL_UNI07_Master.udtMBData			:= udtMbDataMaster;
MB_IL_UNI07_Master.arrInputAddress		:= arrInputAddressMaster;
MB_IL_UNI07_Master.arrOutputAddress		:= arrOutputAddressMaster;

MB_IL_UNI07_Master();

udtMbDataMaster							:= MB_IL_UNI07_Master.udtMBData;
arrInputAddressMaster					:= MB_IL_UNI07_Master.arrInputAddress;
arrOutputAddressMaster					:= MB_IL_UNI07_Master.arrOutputAddress;

(*	FC3 = Read multiple holding registers *)
MB_RTU_FC3.xActivate					:= MB_IL_UNI07_Master.xActive;
MB_RTU_FC3.xSendRequest					:= ModbusControl.xSendRequest_FC3;
MB_RTU_FC3.xEnablePoll					:= FALSE;
MB_RTU_FC3.uiSlaveAddress				:= ModbusControl.uiSlaveAddress;
MB_RTU_FC3.uiStartAddress				:= ModbusControl.uiStartAddress_FC3;
MB_RTU_FC3.iDataCount					:= ModbusControl.iDataCount_FC3;
MB_RTU_FC3.arrReadData					:= ModbusControl.arrReadData_FC3;
MB_RTU_FC3.udtMbData					:= udtMbDataMaster;

MB_RTU_FC3();

ModbusControl.xDone_FC3					:= MB_RTU_FC3.xDone;
ModbusControl.xError_FC3				:= MB_RTU_FC3.xError;
wDiagCodeFC3							:= MB_RTU_FC3.wDiagCode;
wAddDiagCodeFC3							:= MB_RTU_FC3.wAddDiagCode;

ModbusControl.arrReadData_FC3			:= MB_RTU_FC3.arrReadData;
udtMbDataMaster							:= MB_RTU_FC3.udtMbData;

ModbusControl.Master_iFunctionCode		:= udtMbDataMaster.iFunctionCode;
ModbusControl.Master_uiRcvDataCount		:= udtMbDataMaster.uiRcvdDataCount;
ModbusControl.Master_uiSlaveAddress		:= udtMbDataMaster.uiSlaveAddress;
ModbusControl.Master_uiStartAddress		:= udtMbDataMaster.uiStartAddress;

(*	FC6 = Write holding register*)
MB_RTU_FC6.xActivate					:= MB_IL_UNI07_Master.xActive;
MB_RTU_FC6.xSendRequest					:= ModbusControl.xSendRequest_FC6;
MB_RTU_FC6.xEnablePoll					:= FALSE;
MB_RTU_FC6.uiSlaveAddress				:= ModbusControl.uiSlaveAddress;
MB_RTU_FC6.uiStartAddress				:= ModbusControl.uiStartAddress_FC6;
MB_RTU_FC6.wValue						:= ModbusControl.wValue_FC6;
MB_RTU_FC6.udtMbData					:= udtMbDataMaster;

MB_RTU_FC6();

ModbusControl.xDone_FC6				    := MB_RTU_FC6.xDone;
ModbusControl.xError_FC6				:= MB_RTU_FC6.xError;
wDiagCodeFC3							:= MB_RTU_FC6.wDiagCode;
wAddDiagCodeFC3							:= MB_RTU_FC6.wAddDiagCode;

udtMbDataMaster							:= MB_RTU_FC6.udtMbData;

(*@KEY@: END_WORKSHEET *)
(*@KEY@: WORKSHEET
NAME: MockMasterModule
IEC_LANGUAGE: ST
*)
(*	IB IL RS UNI (Proceess data 7 words) software replacement *)
IB_IL_RS_UNI_07_Master.xConsoleLog		:= xDebug;
IB_IL_RS_UNI_07_Master.strConsoleId		:= 'MAS';
IB_IL_RS_UNI_07_Master.udtRS485Line		:= udtRS485Line;
IB_IL_RS_UNI_07_Master.arrInputAddress	:= arrOutputAddressMaster;
IB_IL_RS_UNI_07_Master.arrOutputAddress	:= arrInputAddressMaster;

IB_IL_RS_UNI_07_Master();

udtRS485Line							:= IB_IL_RS_UNI_07_Master.udtRS485Line;
arrOutputAddressMaster					:= IB_IL_RS_UNI_07_Master.arrInputAddress;
arrInputAddressMaster					:= IB_IL_RS_UNI_07_Master.arrOutputAddress;

(*@KEY@: END_WORKSHEET *)
(*@KEY@: WORKSHEET
NAME: Devices
IEC_LANGUAGE: ST
*)
(* ModbusDeviceHandler01	*)
ModbusDeviceHandler01.xActivate				:= xActivate01;
ModbusDeviceHandler01.xSendRequest_IN		:= xStartOfPoll;
ModbusDeviceHandler01.uiSlaveAddress		:= UINT#01;
ModbusDeviceHandler01.ModbusDeviceData		:= ModbusDeviceData01;
ModbusDeviceHandler01.tTimeout				:= T#2S;
ModbusDeviceHandler01.udtModbusControl		:= ModbusControl;

ModbusDeviceHandler01();

ModbusDeviceData01							:= ModbusDeviceHandler01.ModbusDeviceData;
ModbusControl								:= ModbusDeviceHandler01.udtModbusControl;

xConnectionBroken01							:= ModbusDeviceHandler01.xConnectionBroken;
diTimeDiff01								:= ModbusDeviceHandler01.diTimeDiff;
iRtcData01									:= ModbusDeviceData01.DataValues.iRtcMinutes;

(* ModbusDeviceHandler02	*)
ModbusDeviceHandler02.xActivate				:= xActivate02;
ModbusDeviceHandler02.xSendRequest_IN		:= ModbusDeviceHandler01.xSendRequest_OUT;
ModbusDeviceHandler02.uiSlaveAddress		:= UINT#02;
ModbusDeviceHandler02.ModbusDeviceData		:= ModbusDeviceData02;
ModbusDeviceHandler02.tTimeout				:= T#2S;
ModbusDeviceHandler02.udtModbusControl		:= ModbusControl;

ModbusDeviceHandler02();

ModbusDeviceData02							:= ModbusDeviceHandler02.ModbusDeviceData;
ModbusControl								:= ModbusDeviceHandler02.udtModbusControl;

xConnectionBroken02							:= ModbusDeviceHandler02.xConnectionBroken;
diTimeDiff02								:= ModbusDeviceHandler02.diTimeDiff;
iRtcData02									:= ModbusDeviceData02.DataValues.iRtcMinutes;

(*	End of device bus*)
xEndOfPoll									:= ModbusDeviceHandler02.xSendRequest_OUT;

(*@KEY@: END_WORKSHEET *)
END_PROGRAM

(* ---- MockDevices.ST ---- *)
(*@PROPERTIES_EX@
TYPE: POU
LOCALE: 0
IEC_LANGUAGE: ST
PLC_TYPE: independent
PROC_TYPE: independent
*)
(*@KEY@:DESCRIPTION*)

(*@KEY@:END_DESCRIPTION*)
PROGRAM MockDevices

(*Group:Slaves*)

VAR
	SlaveDevice_01 :	SlaveDevice;
	SlaveDevice_02 :	SlaveDevice;
	xActivateSlave01 :	BOOL := TRUE;
	xActivateSlave02 :	BOOL := TRUE;
END_VAR

(*Group:Global*)

VAR_EXTERNAL
	udtRS485Line :	udtRS485Frame;
END_VAR

VAR
	xDebug :	BOOL;
END_VAR

(*@KEY@: WORKSHEET
NAME: MockDevices
IEC_LANGUAGE: ST
*)
(*	Slave 01 *)
SlaveDevice_01.xActivate		:= xActivateSlave01;
SlaveDevice_01.xDebug			:= xDebug;
SlaveDevice_01.strConsoleId		:= 'SLV_01';
SlaveDevice_01.uiSlaveAddress	:= UINT#01;
SlaveDevice_01.udtRS485Line		:= udtRS485Line;

SlaveDevice_01();

udtRS485Line					:= SlaveDevice_01.udtRS485Line;

(*	Slave 02 *)
SlaveDevice_02.xActivate		:= xActivateSlave02;
SlaveDevice_02.xDebug			:= xDebug;
SlaveDevice_02.strConsoleId		:= 'SLV_02';
SlaveDevice_02.uiSlaveAddress	:= UINT#02;
SlaveDevice_02.udtRS485Line		:= udtRS485Line;

SlaveDevice_02();

udtRS485Line					:= SlaveDevice_02.udtRS485Line;

(*@KEY@: END_WORKSHEET *)
END_PROGRAM
